// TIA Portal V20 export
TYPE "UDT_typeSpdCtrl"
   STRUCT
      input : Struct
         bo_enable : Bool := false;
         bo_estop : Bool := false;
         bo_reset : Bool := false;
         r32_speedSet : Real := 0.0;
         r32_torqueLimitSet : Real;
         r32_filterTime : Real := 100.0;
         tCycle : Real := 10.0;
         OBNum : Int := 30;
         HW_IO : HW_IO := 0;
         HW_IO_ADD : HW_IO;
         Reference : Struct
            r32_speed_Rpm : Real;
            r32_Torque_Nm : Real;
            r32_current_A : Real;
            r32_DCVolagte_V : Real;
            r32_power_Kw : Real;
            "r32_temperature_℃" : Real;
         END_STRUCT;
      END_STRUCT;
      output : Struct
         bo_enabled : Bool := false;
         bo_ready : Bool := false;
         bo_driveError : Bool := false;
         r32_actSpeed_Rpm : Real := 0.0;
         r32_actTorque_Nm : Real;
         r32_actCurrent_A : Real;
         r32_actDCVolagte_V : Real;
         r32_actPower_Kw : Real;
         "r32_actTemperature_℃" : Real;
         i16_warningCode : Word;
         i16_faultCode : Word;
      END_STRUCT;
   END_STRUCT;
END_TYPE
